% RSLogix 500 project Board Counter.RSS, saved by version 7.00.00.19 %
PROJECT "TENENCTR"    % processor: MicroLogix 1000 %

PROGRAM FILES
  LAD 2 "MAIN_PROG"  6 rungs
  LAD 3 "BOARD CNT"  4 rungs
  LAD 4 "HMI"  7 rungs
  LAD 5, 6, 7, 8, 9, 10, 11, 12, 13, 14, 15, 16: only END

DATA FILES
  O0 OUTPUT  1 elements
  I1 INPUT  2 elements
  S2 STATUS  33 elements
  B3 BINARY  32 elements
  T4 TIMER  40 elements
  C5 COUNTER  32 elements
  R6 CONTROL  16 elements
  N7 INTEGER  105 elements

LADDER 2 "MAIN_PROG"
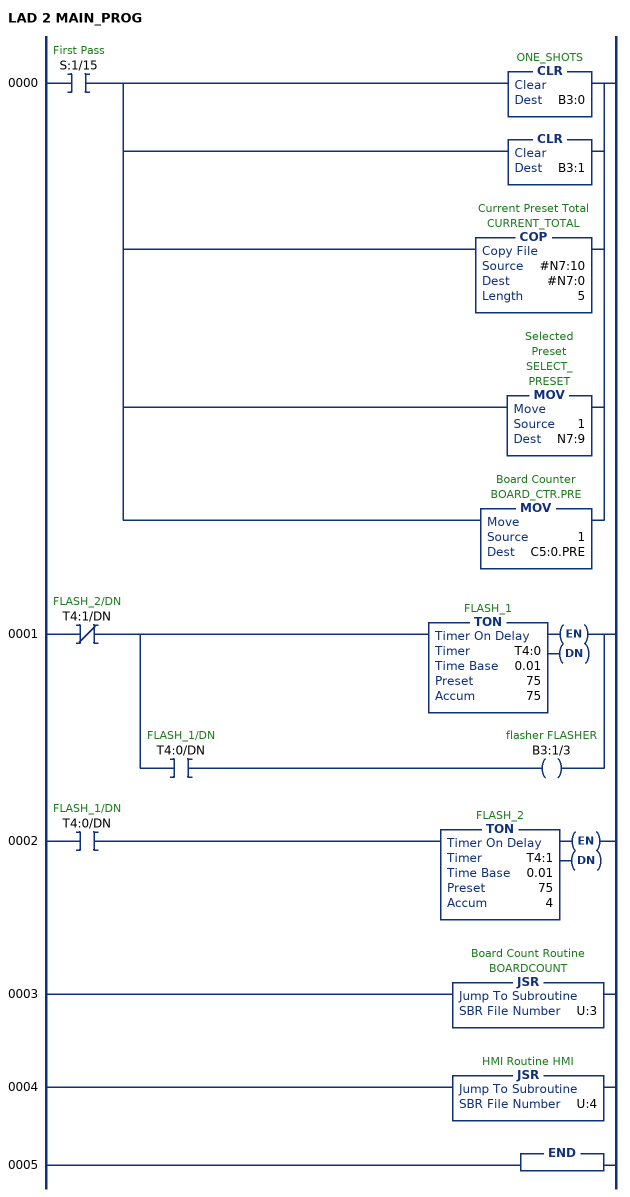
% Rung: 0 %
SOR XIC S:1/15 BST CLR B3:0 NXB CLR B3:1 NXB COP #N7:10 #N7:0 5 NXB MOV 1 N7:9 NXB MOV 1 C5:0.PRE BND EOR
%   S:1/15  "First Pass" %
%   B3:0  ONE_SHOTS %
%   N7:10  PRESET_1_TOTAL  "Preset 1 Total" %
%   N7:0  CURRENT_TOTAL  "Current Preset Total" %
%   N7:9  SELECT_PRESET  "Selected Preset" %
%   C5:0  BOARD_CTR  "Board Counter" %
% Rung: 1 %
SOR XIO T4:1/DN BST TON T4:0 0.01 75 75 NXB XIC T4:0/DN OTE B3:1/3 BND EOR
%   T4:1  FLASH_2 %
%   T4:0  FLASH_1 %
%   B3:1/3  FLASHER  "flasher" %
% Rung: 2 %
SOR XIC T4:0/DN TON T4:1 0.01 75 4 EOR
%   T4:0  FLASH_1 %
%   T4:1  FLASH_2 %
% Rung: 3 %
SOR JSR U:3 EOR
%   U:3  BOARDCOUNT  "Board Count Routine" %
% Rung: 4 %
SOR JSR U:4 EOR
%   U:4  HMI  "HMI Routine" %
% Rung: 5 %
SOR END EOR

LADDER 3 "BOARD CNT"
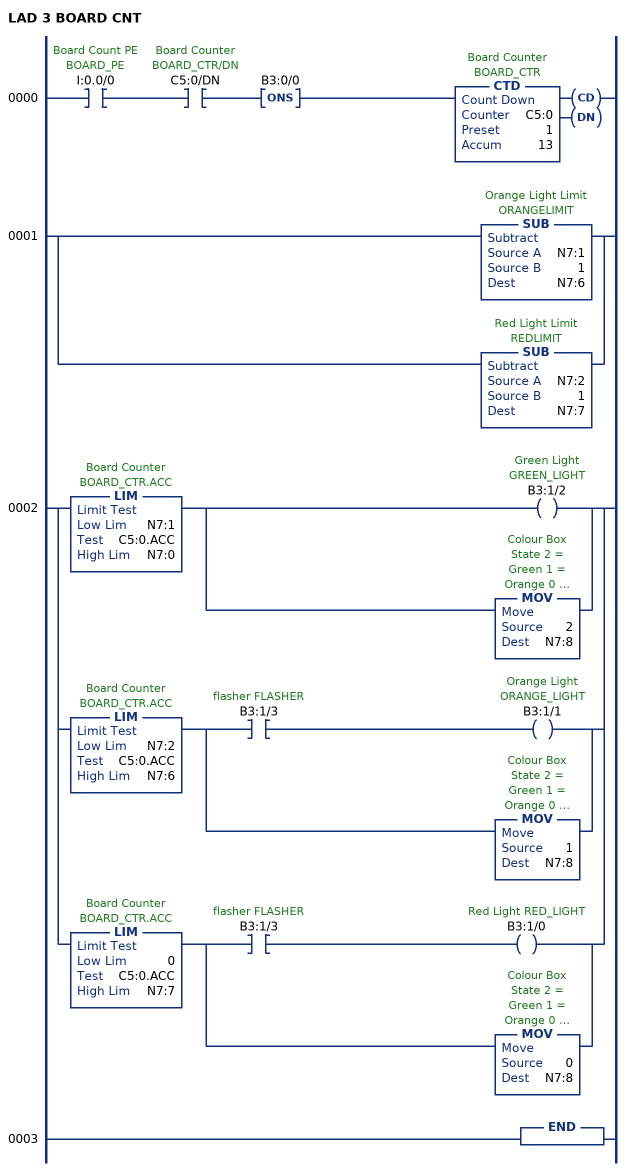
% Rung: 0 %
SOR XIC I:0.0/0 XIC C5:0/DN OSR B3:0/0 CTD C5:0 1 13 EOR
%   I:0.0/0  BOARD_PE  "Board Count PE" %
%   C5:0  BOARD_CTR  "Board Counter" %
% Rung: 1 %
SOR BST SUB N7:1 1 N7:6 NXB SUB N7:2 1 N7:7 BND EOR
%   N7:1  CURRENT_ORN  "Current Preset Orange" %
%   N7:6  ORANGELIMIT  "Orange Light Limit" %
%   N7:2  CURRENT_RED  "Current preset red" %
%   N7:7  REDLIMIT  "Red Light Limit" %
% Rung: 2 %
SOR BST LIM N7:1 C5:0.ACC N7:0 BST OTE B3:1/2 NXB MOV 2 N7:8 BND NXB LIM N7:2 C5:0.ACC N7:6 BST XIC B3:1/3 OTE B3:1/1 NXB MOV 1 N7:8 BND NXB LIM 0 C5:0.ACC N7:7 BST XIC B3:1/3 OTE B3:1/0 NXB MOV 0 N7:8 BND BND EOR
%   N7:1  CURRENT_ORN  "Current Preset Orange" %
%   C5:0  BOARD_CTR  "Board Counter" %
%   N7:0  CURRENT_TOTAL  "Current Preset Total" %
%   B3:1/2  GREEN_LIGHT  "Green Light" %
%   N7:8  COLOUR_BOX_STATE  "Colour Box State 2 = Green 1 = Orange 0 = Red" %
%   N7:2  CURRENT_RED  "Current preset red" %
%   N7:6  ORANGELIMIT  "Orange Light Limit" %
%   B3:1/3  FLASHER  "flasher" %
%   B3:1/1  ORANGE_LIGHT  "Orange Light" %
%   N7:7  REDLIMIT  "Red Light Limit" %
%   B3:1/0  RED_LIGHT  "Red Light" %
% Rung: 3 %
SOR END EOR

LADDER 4 "HMI"
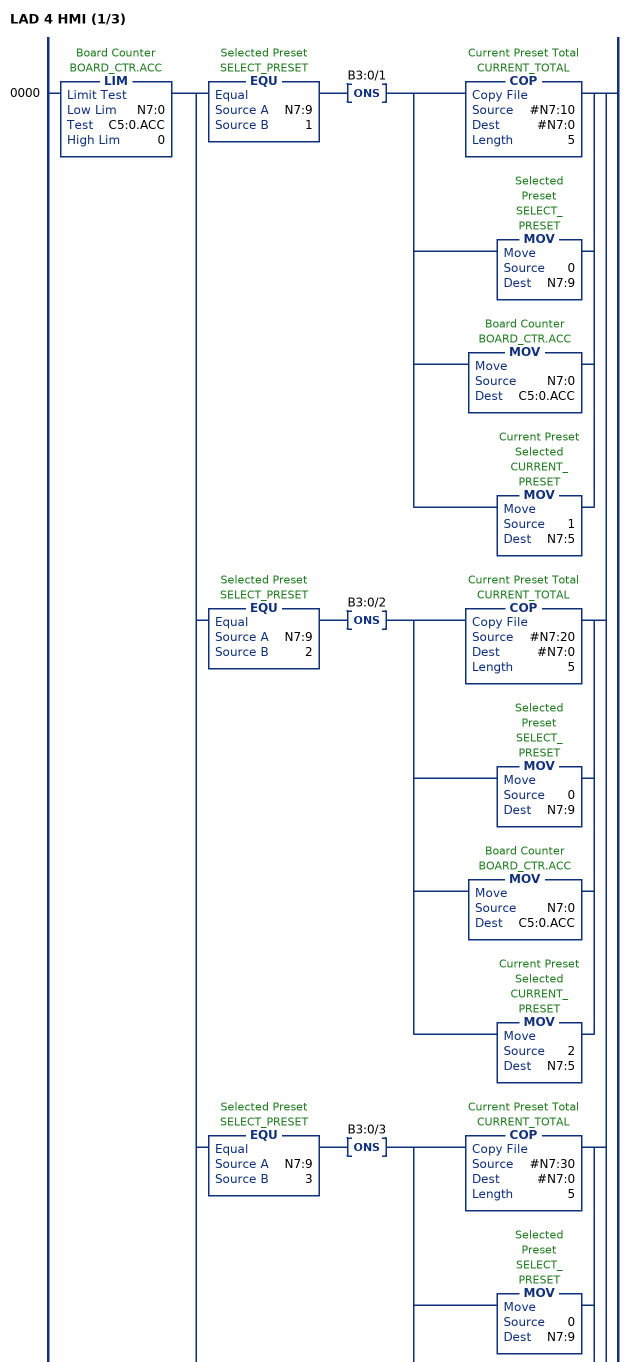
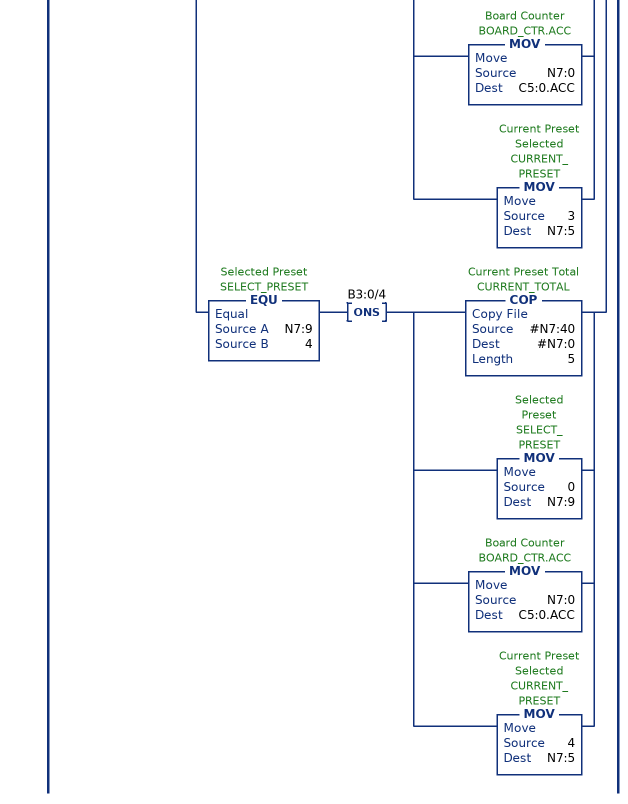
% Rung: 0 %
SOR LIM N7:0 C5:0.ACC 0 BST EQU N7:9 1 OSR B3:0/1 BST COP #N7:10 #N7:0 5 NXB MOV 0 N7:9 NXB MOV N7:0 C5:0.ACC NXB MOV 1 N7:5 BND NXB EQU N7:9 2 OSR B3:0/2 BST COP #N7:20 #N7:0 5 NXB MOV 0 N7:9 NXB MOV N7:0 C5:0.ACC NXB MOV 2 N7:5 BND NXB EQU N7:9 3 OSR B3:0/3 BST COP #N7:30 #N7:0 5 NXB MOV 0 N7:9 NXB MOV N7:0 C5:0.ACC NXB MOV 3 N7:5 BND NXB EQU N7:9 4 OSR B3:0/4 BST COP #N7:40 #N7:0 5 NXB MOV 0 N7:9 NXB MOV N7:0 C5:0.ACC NXB MOV 4 N7:5 BND BND EOR
%   N7:0  CURRENT_TOTAL  "Current Preset Total" %
%   C5:0  BOARD_CTR  "Board Counter" %
%   N7:9  SELECT_PRESET  "Selected Preset" %
%   N7:10  PRESET_1_TOTAL  "Preset 1 Total" %
%   N7:5  CURRENT_PRESET  "Current Preset Selected" %
%   N7:20  PRESET_2_TOTAL  "Preset 2 Total" %
%   N7:30  PRESET_3_TOTAL  "Preset 3 Total" %
%   N7:40  PRESET_4_TOTAL  "Preset 4 Total" %

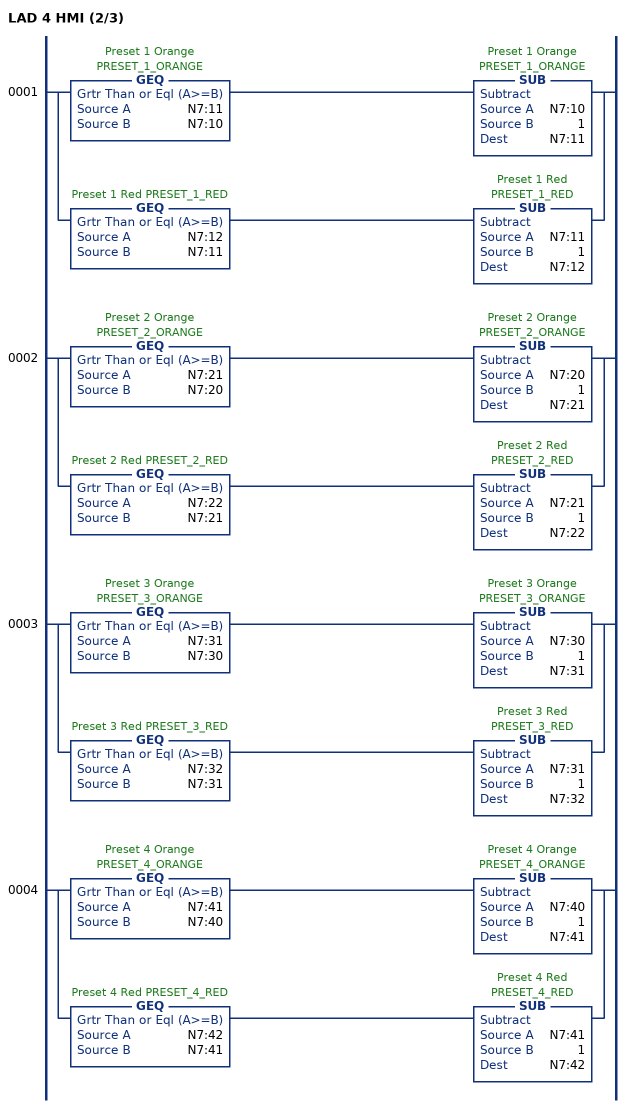
% Rung: 1 %
SOR BST GEQ N7:11 N7:10 SUB N7:10 1 N7:11 NXB GEQ N7:12 N7:11 SUB N7:11 1 N7:12 BND EOR
%   N7:11  PRESET_1_ORANGE  "Preset 1 Orange" %
%   N7:10  PRESET_1_TOTAL  "Preset 1 Total" %
%   N7:12  PRESET_1_RED  "Preset 1 Red" %
% Rung: 2 %
SOR BST GEQ N7:21 N7:20 SUB N7:20 1 N7:21 NXB GEQ N7:22 N7:21 SUB N7:21 1 N7:22 BND EOR
%   N7:21  PRESET_2_ORANGE  "Preset 2 Orange" %
%   N7:20  PRESET_2_TOTAL  "Preset 2 Total" %
%   N7:22  PRESET_2_RED  "Preset 2 Red" %
% Rung: 3 %
SOR BST GEQ N7:31 N7:30 SUB N7:30 1 N7:31 NXB GEQ N7:32 N7:31 SUB N7:31 1 N7:32 BND EOR
%   N7:31  PRESET_3_ORANGE  "Preset 3 Orange" %
%   N7:30  PRESET_3_TOTAL  "Preset 3 Total" %
%   N7:32  PRESET_3_RED  "Preset 3 Red" %
% Rung: 4 %
SOR BST GEQ N7:41 N7:40 SUB N7:40 1 N7:41 NXB GEQ N7:42 N7:41 SUB N7:41 1 N7:42 BND EOR
%   N7:41  PRESET_4_ORANGE  "Preset 4 Orange" %
%   N7:40  PRESET_4_TOTAL  "Preset 4 Total" %
%   N7:42  PRESET_4_RED  "Preset 4 Red" %

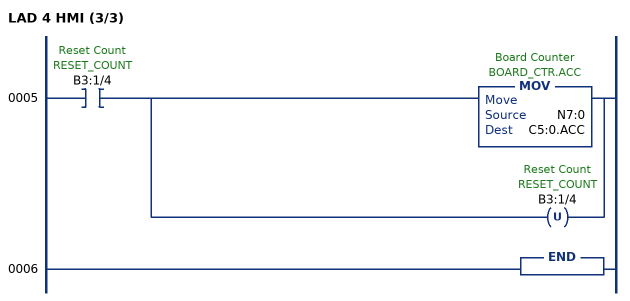
% Rung: 5 %
SOR XIC B3:1/4 BST MOV N7:0 C5:0.ACC NXB OTU B3:1/4 BND EOR
%   B3:1/4  RESET_COUNT  "Reset Count" %
%   N7:0  CURRENT_TOTAL  "Current Preset Total" %
%   C5:0  BOARD_CTR  "Board Counter" %
% Rung: 6 %
SOR END EOR

DATA TABLE (non-zero values as saved)
DATA B3
% B3:0 % 0X0000 0X0004 0X0000 0X0000 0X0000 0X0000 0X0000 0X0000 0X0000 0X0000
DATA T4
% .PRE .ACC %
% T4:0 % 75 75
% T4:1 % 75 4
DATA C5
% .PRE .ACC %
% C5:0 % 1 13
DATA N7
% N7:0 % 13 3 925 0 0 0 2 924 0 0
% N7:10 % 13 3 2 0 0 0 0 0 0 0
% N7:20 % 34 33 0 0 0 0 0 0 0 0
% N7:30 % 20 12 2 0 0 0 0 0 0 0
% N7:40 % 20 14 2 0 0 0 0 0 0 0
